Universal Robots PolyScope program: RC_E7_MOVE_710.urp

Program RC_E7_MOVE_710 (createdIn=3.0.0 lastSavedIn=3.0.0 directory=/programs installation=default)
Robot Program (runOnlyOnce=true motionType=MoveJ speed=1.047198 acceleration=1.396263 useActiveTCP=false)
  'Program generated by RoboDK v4.1.0 for UR3e_HORNO on 05/09/2022 13:22:10'
  'Using nominal kinematics.'
  'Using Ref. UR3_2: p[0.000000, 0.000000, 0.000000, 0.000000, 0.000000, 0.000000]'
  'Using TCP 0208-0001-0001-307-000-3 Horno: p[0.000000, 0.000000, 0.164750, 0.000000, 0.000000, 0.000000]'
  Script: set_tcp(p[0.000000, 0.000000, 0.164750, 0.000000, 0.000000, 0.000000])
  Script: movej([-0.742110, -1.409854, -0.955499, -2.344942, 1.570617, 0.000004],0.60000,0.12500,0,0.0000)
